{attribute 'GeneratedUsingTerminal: EL2595-0000-0018'}
{attribute addProperty BoxType "EL2595-0000-0018"}
{attribute addProperty Id "Ready_to_activateBOOL1Output_activeBOOL1WarningBOOL1ErrorBOOL1Digital_inputBOOL1TxPDO_ToggleBOOL1"}
{attribute addProperty CRC "1005865601"}
{attribute addProperty Size "6"}
TYPE Status_3BF44A81 :
STRUCT
	{attribute addProperty Name "Ready_to_activate"}
	Ready_to_activate : BOOL;
	{attribute addProperty Name "Output_active"}
	Output_active : BOOL;
	{attribute addProperty Name "Warning"}
	Warning : BOOL;
	{attribute addProperty Name "Error"}
	Error : BOOL;
	{attribute addProperty Name "Digital_input"}
	Digital_input : BOOL;
	{attribute addProperty Name "TxPDO_Toggle"}
	TxPDO_Toggle : BOOL;
END_STRUCT
END_TYPE

(* stored: Version 1.2.0.0, ProductVersion 3.1.4024.11
   DUT Status_3BF44A81: Id {41bf9509-18d2-4254-a0d4-4ab81acb26e3} *)
